PROGRAM MAIN
VAR
	bStartMotor : BOOL := FALSE;
	bStopMotor  : BOOL := FALSE;
	bServoMotor : BOOL;
	sr_MotorSetReset : SR;
END_VAR


sr_MotorSetReset(SET1:= bStartMotor,
				 RESET:= bStopMotor,
				 Q1 => bServoMotor);

p10_ladder();

END_PROGRAM

(* stored: Version 1.1.0.1, ProductVersion 3.1.4024.13
   POU MAIN: Id {b6d9fbc8-18d9-4327-b2b8-220f27d5c483}, SpecialFunc None *)
